TYPE csp_case_phasing_enum :
(
	CSP_CASE_PHASING_START							:= 1,
	//CSP_CASE_PHASING_CHECK_ALL_INTERFERENCE			:= 10,
	CSP_CASE_PHASING_CHECK_LEADING_MINOR			:= 20,
	CSP_CASE_PHASING_CHECK_LOADER_GUIDES			:= 30,
	CSP_CASE_PHASING_CHECK_LOADER					:= 40,
	CSP_CASE_PHASING_CHECK_FOLLOWER					:= 50,
	
	CSP_CASE_PHASING_MOVE_GUIDES					:= 100,
	CSP_CASE_PHASING_REORDER_GUIDES					:= 105,
	CSP_CASE_PHASING_MOVE_DOWNSTREAM_GUIDE			:= 110,
	CSP_CASE_PHASING_MOVE_DOWNSTREAM_GUIDE_OUT		:= 115,
	CSP_CASE_PHASING_MOVE_UPSTREAM_GUIDE			:= 120,
	CSP_CASE_PHASING_MOVE_UPSTREAM_GUIDE_OUT		:= 125,
	CSP_CASE_PHASING_GUIDES_OUT						:= 127,
	CSP_CASE_PHASING_GUIDE_MOVE_COMPLETE			:= 130,
	
	CSP_CASE_PHASING_MOVE_LOADER					:= 200,
	CSP_CASE_PHASING_MOVE_LOADER_COMPLETE			:= 210,
	
	CSP_CASE_PHASING_MOVE_FOLLOWER					:= 300,
	CSP_CASE_PHASING_MOVE_FOLLOWER_COMPLETE			:= 310,
	
	CSP_CASE_PHASING_DONE							:= 900,
	CSP_CASE_PHASING_ERROR							:= 999
) := CSP_CASE_PHASING_DONE;
END_TYPE

(* stored: Version 1.1.0.1, ProductVersion 3.1.4024.3
   DUT csp_case_phasing_enum: Id {20edd24c-118c-057b-199a-3b3a62eee049} *)
